Yaskawa INFORM job: MALBEN5.JBI

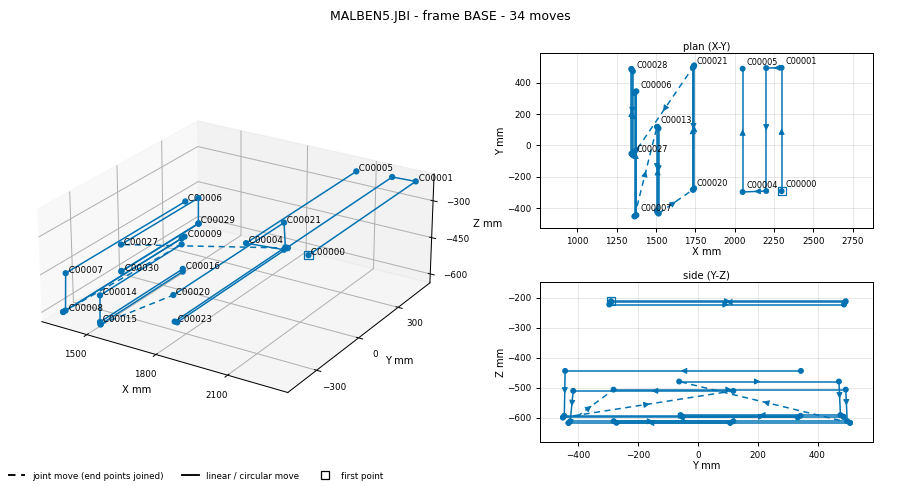
[picture p0: tool path of MALBEN5.JBI in frame BASE, 34 of 40 moves have a stored position in this frame; points joined in program order, loops and branches not executed]
/JOB
//NAME MALBEN5
//POS
///NPOS 34,0,34,0,0,0
///TOOL 0
///POSTYPE BASE
///RECTAN
///RCONF 1,0,0,0,0,0,0,0,0,0,0,0,0,0,0,0,0,0,0,0,0,0,0,0
C00000=2298.803439,-290.558510,-210.984393,175.000000,5.000000,5.000000
C00001=2298.803439,494.294586,-210.984393,175.000000,5.000000,5.000000
C00002=2200.866433,492.764092,-214.105643,175.000000,5.000000,5.000000
C00003=2200.866433,-289.515320,-214.105643,175.000000,5.000000,5.000000
C00004=2050.856817,-296.008692,-222.209152,175.000000,5.000000,5.000000
C00005=2050.856817,488.444031,-222.209152,175.000000,5.000000,5.000000
C00006=1375.075213,344.427756,-444.002571,175.000000,-89.999999,5.000000
C00007=1375.075213,-443.698830,-444.002571,175.000000,-89.999999,5.000000
C00008=1370.457012,-446.399049,-594.002571,175.000000,-89.999999,5.000000
C00009=1370.457012,343.178827,-594.002571,175.000000,-89.999999,5.000000
C00010=1363.109600,333.694012,-599.665004,180.000000,-60.000000,0.000000
C00011=1363.109600,-450.921951,-599.665004,180.000000,-60.000000,0.000000
C00012=1363.109600,-450.921951,-599.665004,180.000000,-60.000000,0.000000
C00013=1505.777973,118.607127,-510.797933,175.000000,-89.999999,5.000000
C00014=1505.777973,-416.713173,-510.797933,175.000000,-89.999999,5.000000
C00015=1509.734888,-426.727448,-612.380156,175.000000,-89.999999,5.000000
C00016=1509.734888,118.634509,-612.380156,175.000000,-89.999999,5.000000
C00017=1516.209668,107.922922,-618.042589,180.000000,-60.000000,0.000000
C00018=1516.209668,-432.333933,-618.042589,180.000000,-60.000000,0.000000
C00019=1516.209668,-432.333933,-618.042589,180.000000,-60.000000,0.000000
C00020=1733.696846,-281.738164,-506.566317,175.000000,-89.999999,5.000000
C00021=1733.696846,494.416615,-506.566317,175.000000,-89.999999,5.000000
C00022=1737.814807,499.280727,-611.960853,175.000000,-89.999999,5.000000
C00023=1737.814807,-281.354937,-611.960853,175.000000,-89.999999,5.000000
C00024=1742.590608,-272.126332,-617.623286,180.000000,-60.000000,0.000000
C00025=1742.590608,508.707587,-617.623286,180.000000,-60.000000,0.000000
C00026=1742.590608,508.707587,-617.623286,180.000000,-60.000000,0.000000
C00027=1352.721148,-62.507450,-479.553261,175.000000,-89.999999,5.000000
C00028=1352.721148,471.579930,-479.553261,175.000000,-89.999999,5.000000
C00029=1348.526463,476.738273,-591.716491,175.000000,-89.999999,5.000000
C00030=1348.526463,-57.713278,-591.716491,175.000000,-89.999999,5.000000
C00031=1343.112300,-51.728627,-597.378924,180.000000,-60.000000,0.000000
C00032=1343.112300,486.733989,-597.378924,180.000000,-60.000000,0.000000
C00033=1343.112300,486.733989,-597.378924,180.000000,-60.000000,0.000000
///POSTYPE PULSE
///PULSE
EC00000=0
EC00001=0
EC00002=0
EC00003=0
EC00004=0
EC00005=0
EC00006=0
EC00007=0
EC00008=0
EC00009=0
EC00010=0
EC00011=0
EC00012=92160
EC00013=92160
EC00014=92160
EC00015=92160
EC00016=92160
EC00017=92160
EC00018=92160
EC00019=184320
EC00020=184320
EC00021=184320
EC00022=184320
EC00023=184320
EC00024=184320
EC00025=184320
EC00026=276480
EC00027=276480
EC00028=276480
EC00029=276480
EC00030=276480
EC00031=276480
EC00032=276480
EC00033=368640
//INST
///DATE 2023/04/20 17:25
///ATTR SC,RW,RJ
////FRAME BASE
///GROUP1 RB1,ST1
NOP
MOVJ P009 EX000 VJ=15.00
MOVJ C00000 EC00000 VJ=15.0
CALL JOB:SPYON
MOVL C00001 EC00001 V=200.0
MOVL C00002 EC00002 V=200.0
MOVL C00003 EC00003 V=200.0
MOVL C00004 EC00004 V=200.0
MOVL C00005 EC00005 V=200.0
CALL JOB:SPYOF
MOVJ P009 VJ=15.00
MOVJ C00006 EC00006 VJ=15.0
CALL JOB:SPYON
MOVL C00007 EC00007 V=200.0
MOVL C00008 EC00008 V=200.0
MOVL C00009 EC00009 V=200.0
MOVL C00010 EC00010 V=200.0
MOVL C00011 EC00011 V=200.0
CALL JOB:SPYOF
MOVJ P009 VJ=15.00
MOVL C00012 EC00012 V=200.0
MOVJ C00013 EC00013 VJ=15.0
CALL JOB:SPYON
MOVL C00014 EC00014 V=200.0
MOVL C00015 EC00015 V=200.0
MOVL C00016 EC00016 V=200.0
MOVL C00017 EC00017 V=200.0
MOVL C00018 EC00018 V=200.0
CALL JOB:SPYOF
MOVJ P009 VJ=15.00
MOVL C00019 EC00019 V=200.0
MOVJ C00020 EC00020 VJ=15.0
CALL JOB:SPYON
MOVL C00021 EC00021 V=200.0
MOVL C00022 EC00022 V=200.0
MOVL C00023 EC00023 V=200.0
MOVL C00024 EC00024 V=200.0
MOVL C00025 EC00025 V=200.0
CALL JOB:SPYOF
MOVJ P009 VJ=15.00
MOVL C00026 EC00026 V=200.0
MOVJ C00027 EC00027 VJ=15.0
CALL JOB:SPYON
MOVL C00028 EC00028 V=200.0
MOVL C00029 EC00029 V=200.0
MOVL C00030 EC00030 V=200.0
MOVL C00031 EC00031 V=200.0
MOVL C00032 EC00032 V=200.0
CALL JOB:SPYOF
MOVJ P009 VJ=15.00
MOVL C00033 EC00033 V=200.0
END
